FUNCTION F_SAFETY_StatusFB_TO_DECOUPLE : ST_SAFETY_FBDECOUPLE
VAR_INPUT
	stFBStatus						: ST_SAFETY_FBStatus; 	(* Struktura ogolna *)
END_VAR

F_SAFETY_StatusFB_TO_DECOUPLE.uStatus.stStatusWords 		:= stFBStatus;					(* Przepisanie *)
F_SAFETY_StatusFB_TO_DECOUPLE.eState					 	:= stFBStatus.BState;			(* Ustawienie enum *)

END_FUNCTION

(* stored: Version 1.1.0.1, ProductVersion 3.1.4022.12
   POU F_SAFETY_StatusFB_TO_DECOUPLE: Id {691277ce-41df-43ee-b7f1-bceff6da647c}, SpecialFunc None *)
